# EPICS substitutions: mc10/tpmacApp/Db/autohome.substitutions
file "$(EPICS_BASE)/db/autohome.db"
{

pattern
{SYS,              DEV,                 PLC,  PORT  }
{"XF:23ID1-OP",  "{Slt:3-Ax:Y}",      8 ,     P0    }
{"XF:23ID1-OP",  "{Slt:3-Ax:X}",      9 ,     P0    }
{"XF:23ID1-ES",  "{Cam:Beam-Ax:X}",      10 ,     P0    }
{"XF:23ID1-ES",  "{Cam:Beam-Ax:Z}",      11 ,    P0    }
{"XF:23ID1-ES",  "{Cam:Beam-Ax:Zm}",      13 ,    P0    }
{"XF:23ID1-ES",  "{Cam:Beam-Ax:Foc}",      12 ,    P0    }

}
